# EPICS autosave request: iocs/SIS8300bpmIOC/iocBoot/iocSIS8300bpm/auto_settings.req
file "SIS8300bpm_settings.req",         P=$(P),  R=
file "SIS8300bpmN_settings.req",        P=$(P),  R=AI1:
file "SIS8300bpmN_settings.req",        P=$(P),  R=AI2:
file "SIS8300bpmN_settings.req",        P=$(P),  R=AI3:
file "SIS8300bpmN_settings.req",        P=$(P),  R=AI4:
file "SIS8300bpmN_settings.req",        P=$(P),  R=AI5:
file "SIS8300bpmN_settings.req",        P=$(P),  R=AI6:
file "SIS8300bpmN_settings.req",        P=$(P),  R=AI7:
file "SIS8300bpmN_settings.req",        P=$(P),  R=AI8:
file "SIS8300bpmN_settings.req",        P=$(P),  R=AI9:
file "SIS8300bpmN_settings.req",        P=$(P),  R=AI10:
file "NDStdArrays_settings.req",     P=$(P),  R=image1:
file "commonPlugin_settings.req",    P=$(P)
file "NDTimeSeries_settings.req",    P=$(P),  R=TS:
file "NDTimeSeriesN_settings.req",   P=$(P),  R=TS:1:
file "NDTimeSeriesN_settings.req",   P=$(P),  R=TS:2:
file "NDTimeSeriesN_settings.req",   P=$(P),  R=TS:3:
file "NDTimeSeriesN_settings.req",   P=$(P),  R=TS:4:
file "NDTimeSeriesN_settings.req",   P=$(P),  R=TS:5:
file "NDTimeSeriesN_settings.req",   P=$(P),  R=TS:6:
file "NDTimeSeriesN_settings.req",   P=$(P),  R=TS:7:
file "NDTimeSeriesN_settings.req",   P=$(P),  R=TS:8:
file "NDTimeSeriesN_settings.req",   P=$(P),  R=TS:9:
file "NDTimeSeriesN_settings.req",   P=$(P),  R=TS:10:
file "NDFFT_settings.req",           P=$(P),  R=FFT1:
file "NDFFT_settings.req",           P=$(P),  R=FFT2:
file "NDFFT_settings.req",           P=$(P),  R=FFT3:
file "NDFFT_settings.req",           P=$(P),  R=FFT4:
file "NDFFT_settings.req",           P=$(P),  R=FFT5:
file "NDFFT_settings.req",           P=$(P),  R=FFT6:
file "NDFFT_settings.req",           P=$(P),  R=FFT7:
file "NDFFT_settings.req",           P=$(P),  R=FFT8:
file "NDFFT_settings.req",           P=$(P),  R=FFT9:
file "NDFFT_settings.req",           P=$(P),  R=FFT10:
